VAR_GLOBAL CONSTANT
	MAX_BUFFER_SIZE : UDINT := 1000;
END_VAR

(* stored: Version 1.1.0.1, ProductVersion 3.1.0.24
   GVL GVL: Id {20d915b3-a1c1-4a4e-beca-3855444214bd} *)
